Staubli VAL3: stop.pgx

program stop()
begin
  //
  disablePower()
  resetMotion()
  libSave()
  cls()
  popUpMsg("程序结束")
  call killAllTask()
end
